(* CODESYS project CmpTemplateEventIECTest.project

Project tree, tasks and I/O mapping:
  Device : CODESYS Control Win V3, 3S - Smart Software Solutions GmbH, order no. 305021, version 3.5.8.0
    application Application
      libraries: Standard, * (System); CmpEventMgr, 3.5.8.0 (System); SysTypes Interfaces, * (System); CmpLog, * (System); CmpErrors Interfaces, * (System); CoDeSys Event Usage Template, 3.5.8.0 (3S - Smart Software Solutions GmbH)
      task MainTask (cyclic, interval t#20ms, priority 1) calls PLC_PRG
      program PLC_PRG [ST]
      function MyCallbackFunction [ST]
      global variables GVL
*)

// Device/Application/GVL
VAR_GLOBAL
	// If callback is registered, this variable is increased in every communication cycle of the runtime system
	nEventCount: INT;
	
	// Example to read event parameter. Should be 17 if callback is registered
	dwParam1: DWORD;
END_VAR

// Device/Application/PLC_PRG
PROGRAM PLC_PRG
VAR
	eventTest: RTS_IEC_HANDLE := RTS_INVALID_HANDLE;
	result: RTS_IEC_RESULT;
	bRegister: BOOL;
	bUnRegister: BOOL;
END_VAR

// Set to TRUE to register callback. GVL.nEventCount will start to increment
IF bRegister THEN
	bRegister := FALSE;
	
	// Open the event
	eventTest := EventOpen(EVTDEMO.EVT_Test, EVTDEMO.CmpId_CmpTest, Result);

	IF eventTest = RTS_INVALID_HANDLE THEN
		LogAdd(STD_LOGGER, 'MyIECApplication', UDINT_TO_DINT(LogClass.LOG_ERROR), 17, 4, 'EventOpen failed. Please check if runtime component is included in runtime configuration'); 
	END_IF
	
	// Register the callback
	result := EventRegisterCallbackFunction(eventTest, ADR(MyCallbackFunction));

	IF result <> CmpErrors.Errors.ERR_OK THEN
		LogAdd(STD_LOGGER, 'MyIECApplication', UDINT_TO_DINT(LogClass.LOG_ERROR), 17, 4, 'EventRegisterCallbackFunction failed. ERR_PARAMETER = 0x0002 means invalid event'); 
	END_IF
END_IF

// Set to TRUE to unregister callback. GVL.nEventCount will stop to increment
IF bUnRegister THEN
	bUnRegister := FALSE;

	// UnRegister the callback
	result := EventUnregisterCallbackFunction(eventTest, ADR(MyCallbackFunction));
	
	// Close the event
	result := EventClose2(eventTest);
	eventTest := RTS_INVALID_HANDLE;
END_IF

END_PROGRAM

// Device/Application/MyCallbackFunction
FUNCTION MyCallbackFunction : RTS_IEC_RESULT
VAR_INPUT
	param: POINTER TO EventParam;
END_VAR
VAR
	pEventParam: POINTER TO EVTDEMO.EVTPARAM_EvtTest;
END_VAR

// 
nEventCount := nEventCount + 1;
// 

// Use param^.CmpIdProvider to identify the component that posts the event. Note that param^.EventId is not unique in the system */
CASE param^.CmpIdProvider OF
	EVTDEMO.CmpId_CmpTest:
		// Use param^.EventId to identify the event. 
		CASE param^.EventId OF
			EVTDEMO.EVT_Test:
				// Check usParamId and usVersion to use correct event structure
				IF  param^.usParamId = EVTDEMO.EVTPARAMID_CmpTemplateEventIEC AND param^.usVersion = EVTDEMO.EVTVERSION_CmpTemplateEventIEC THEN
					// Retrieve pointer to specific event parameter
					pEventParam := param^.pParameter;
					// Example, read parameter value and store to global variable
					dwParam1 := pEventParam^.dwParam1;
				END_IF
		END_CASE
END_CASE

END_FUNCTION
